TYPE ST_WeighingBottleParams :
STRUCT
	rTargetWeight: REAL;
	rWeightTolerance: REAL;
	wVisionInspections: WORD;
END_STRUCT
END_TYPE

(* stored: Version 1.1.0.1, ProductVersion 3.1.4024.15
   DUT ST_WeighingBottleParams: Id {508e49c6-b4c4-4c9f-95b1-8d3a68d161a7} *)
